{attribute 'linkalways'} 
{attribute 'no_explicit_call' := 'This FB is a CLASS and must be accessed using methods or properties'}
{attribute 'enable_dynamic_creation'}
FUNCTION_BLOCK FINAL DigitalInputNode EXTENDS Node
VAR
	input AT %I* : BOOL;
	out : _BOOL(FALSE);
END_VAR

METHOD PUBLIC Clone : I_Node
VAR
END_VAR
Clone := this^;
END_METHOD

METHOD Dispose
VAR_INPUT
END_VAR
END_METHOD

METHOD FB_init : BOOL
VAR_INPUT
	bInitRetains : BOOL; // if TRUE, the retain variables are initialized (warm start / cold start)
	bInCopyCode : BOOL;  // if TRUE, the instance afterwards gets moved into the copy code (online change)
END_VAR
AddOutput('out', out);
END_METHOD

METHOD PROTECTED OnExecute : HRESULT
VAR
END_VAR
out.value := input;
END_METHOD

END_FUNCTION_BLOCK

(* stored: Version 1.1.0.1, ProductVersion 3.1.4024.12
   POU DigitalInputNode: Id {5ee06dc0-2d4f-0ec7-1e1c-92a85ff2854f}, SpecialFunc None
   Folder Constructor: Id {56868e72-7ab7-051a-0934-7fbcb45bc037}
   Method Clone: Id {4f4de4e1-56b3-0c4c-3dea-4e1dda933bc0}
   Method Dispose: Id {f2797aac-e6be-08db-2041-402a0468c712}
   Method FB_init: Id {8a4ae604-15d8-0c76-0e11-d9e137dfbbde}
   Method OnExecute: Id {9126a9b0-01b7-0fbf-3580-4b7fea5bc8a1} *)
